KUKA KRL data list: signals_and_timers.dat

&ACCESS RVP
&REL 1
&COMMENT Data list for signals and timers demonstration
DEFDAT signals_and_timers PUBLIC
  DECL GLOBAL REAL rCalibrationFactor = 1.024
ENDDAT
